// TIA Portal V17 export
// export: Created 2023-02-14T02:49:13.954681Z, ExportSetting WithDefaults, DisplayName Totally Integrated Automation Portal, DisplayVersion V17, DisplayName TIA Portal Openness, DisplayVersion V17, DisplayName TIA Portal Teamcenter Gateway, DisplayVersion V17, DisplayName TIA Portal Version Control Interface, DisplayVersion V17, DisplayName SINAMICS Startdrive Advanced, DisplayVersion V17, DisplayName SINAMICS Startdrive G130, G150, S120, S150, SINAMICS MV, S210, DisplayVersion V17, DisplayName SINAMICS Startdrive G110M, G120, G120C, G120D, G120P, G115D, DisplayVersion V17, DisplayName STEP 7 Professional, DisplayVersion V17, DisplayName STEP 7 Safety, DisplayVersion V17, DisplayName WinCC Professional, DisplayVersion V17
DATA_BLOCK "Stock Tank Pouch"   // DB453
{ S7_Optimized_Access := 'FALSE' }
VERSION : 0.1
// stored: AutoNumber false, DBAccessibleFromOPCUA true, DBAccessibleFromWebserver true, IsOnlyStoredInLoadMemory false, IsWriteProtectedInAS false
   VAR RETAIN
      "ST-11 Product Request" : Bool;
      "ST-11 CIP Request" : Bool;
      "ST-14 Product Request" : Bool;
      "ST-14 CIP Request" : Bool;
      "ST-16 Product Request" : Bool;
      "ST-16 CIP Request" : Bool;
      "ST-11_P-81.01 Run" : Bool;
      "ST-14_P-84.01 Run" : Bool;
      "ST-14_P-84.02 Run" : Bool;
      "ST-16_P-82.01 Run" : Bool;
      "ST-14_P-84.01 SP" : Real;
      "ST-14_P-84.02 SP" : Real;
      "ST-16_P-82.01 SP" : Real;
      "ST-14_P-84.01 Act" : Real;
      "ST-14_P-84.02 Act" : Real;
      "ST-16_P-82.01 Act" : Real;
      "Level ST-14" : Real;
      "Level ST-16" : Real;
      "ST-11_P-81.01 SP" : Real;
      "ST-11_P-81.01 Act" : Real;
      "Level ST-11" : Real;
      freeReal12 : Real;
      freeReal13 : Real;
      freeReal14 : Real;
      freeReal15 : Real;
      freeReal16 : Real;
   END_VAR
BEGIN
END_DATA_BLOCK
